// TIA Portal V19 export
DATA_BLOCK "CONTINUE DB"   // DB11
{ S7_Optimized_Access := 'TRUE' }
// stored: MemoryReserve 100
   VAR RETAIN
      "SYRUP MFG PROCESS ERROR" : Int;
      "PREMIXING PROCESS ERROR" : Int;
      "SUGAR PROCESS ERROR" : Int;
      "MFG PROCESS CONTINUE" : Bool;
      "MFG PROCESS RESET" : Bool;
      "PREMIX PROCESS CONTINUE" : Bool;
      "PREMIX PROCESS RESET" : Bool;
      "SUGAR PROCESS CONTINUE" : Bool;
      "SUGAR PREMIX PROCESS RESET" : Bool;
   END_VAR
BEGIN
END_DATA_BLOCK
